DATA_BLOCK "ST10_SystemModeFB_iDB"
VAR
  sRunT : TON_TIME;
  sPressureTOF : TOF_TIME;
  sChangeOverTOF : TOF_TIME;
  sChangeOverOK : Bool;
END_VAR
BEGIN
END_DATA_BLOCK
